FUNCTION_BLOCK FB_PressureTransceiver_Sim EXTENDS FB_PressureSensor
VAR_INPUT
    bPumpIsON : BOOL; // generates signal based on pump input
    simCellState : eCellState;
END_VAR
VAR_OUTPUT
END_VAR
VAR
    signalClimbTON : TON := (PT := T#25MS);
    signalFallTON : TON := (PT := T#50ms);
    
    simPressureDropTON : TON := (PT := T#70S);
END_VAR

IF bPumpIsON AND (curState = eState_Idle) THEN
    // simulate a rising signal when pump is ON
    nextState := eState_Startup;
END_IF

ExecuteState();
IF NOT (nextState = curState)THEN
    StateTransition();
END_IF

ACTION ExecuteState:


CASE curState OF
	eState_Idle: ExecuteState_Idle();
	eState_Startup: ExecuteState_Startup();
	eState_Running: ExecuteState_Running();
	eState_Complete: ExecuteState_Complete();
	eState_Error: ExecuteState_Error();
	eState_Independent: ExecuteState_Independent();
END_CASE
END_ACTION

ACTION ExecuteState_Complete:

END_ACTION

ACTION ExecuteState_Error:

END_ACTION

ACTION ExecuteState_Idle:

END_ACTION

ACTION ExecuteState_Independent:

END_ACTION

ACTION ExecuteState_Running:
IF bPumpIsON THEN

    // psi climbs
    signalClimbTON(IN := TRUE);
    IF signalClimbTON.Q THEN
        fBufferedSignal := fBufferedSignal + 0.1;
        signalClimbTON(IN := FALSE);
    END_IF

ELSE

    // psi falls
    IF fBufferedSignal < 2 THEN // if somehow signal falls below
        fBufferedSignal := 2;
    END_IF
    IF fBufferedSignal > 2 THEN // only if signal is more than hardware min decrease it
        signalFallTON(IN := TRUE);
        IF signalFallTON.Q THEN
            fBufferedSignal := fBufferedSignal - 0.01;
            signalFallTON(IN := FALSE);
        END_IF
	END_IF

END_IF


// every nth seconds simulate a pressure drop error
IF simCellState = eCellState_Automatic OR simCellState = eCellState_Manual THEN
    simPressureDropTON(IN := TRUE);
    IF simPressureDropTON.Q THEN
        fBufferedSignal := 2;
        simPressureDropTON(IN := FALSE);
    END_IF
END_IF
END_ACTION

ACTION ExecuteState_Startup:
// Build up pressure first

nextState := eState_Running;
END_ACTION

METHOD getSignal : LREAL
VAR_INPUT
END_VAR
// return signal value to outside world
getSignal := fBufferedSignal;
END_METHOD

METHOD setSignal : BOOL
VAR_INPUT
    input : LREAL;
END_VAR
fInputSignal := input;
END_METHOD

ACTION StateTransition:
//reset timers

SUPER^.StateTransition();
END_ACTION

END_FUNCTION_BLOCK

(* stored: Version 1.1.0.1, ProductVersion 3.1.4024.9
   POU FB_PressureTransceiver_Sim: Id {59b5bed2-690e-4dc4-8e47-89fe44abd589}, SpecialFunc None
   Folder States: Id {23f1721b-6be5-4c06-97da-ab16425c1119}
   Action ExecuteState: Id {5ae98e6b-9a60-4f9b-a5f8-093aed8e4c6a}
   Action ExecuteState_Complete: Id {dc68b15a-d715-4c4b-93c9-5479110e9dc2}
   Action ExecuteState_Error: Id {d748b74a-867e-463d-b64c-5e1cc7c851d1}
   Action ExecuteState_Idle: Id {079af7d6-c033-4459-9d39-a9f287a5a4d5}
   Action ExecuteState_Independent: Id {ea546268-67db-4795-bfb3-aad8e1d39961}
   Action ExecuteState_Running: Id {8e2ee644-74d5-4ae4-9033-a5dabc1edd00}
   Action ExecuteState_Startup: Id {4ea1d7b5-5cba-40af-8421-79cf0820c282}
   Method getSignal: Id {b6f6ab00-7a39-447b-84ae-33ea9cce26c7}
   Method setSignal: Id {34e3483a-b4a0-4f13-8263-3003bbd89c16}
   Action StateTransition: Id {6ec8632e-e4bb-4075-8cb2-71d1a4af125c} *)
